KUKA KRL program: Rack_Azul_CogerST121N.src, Rack_Azul_CogerST121N.dat

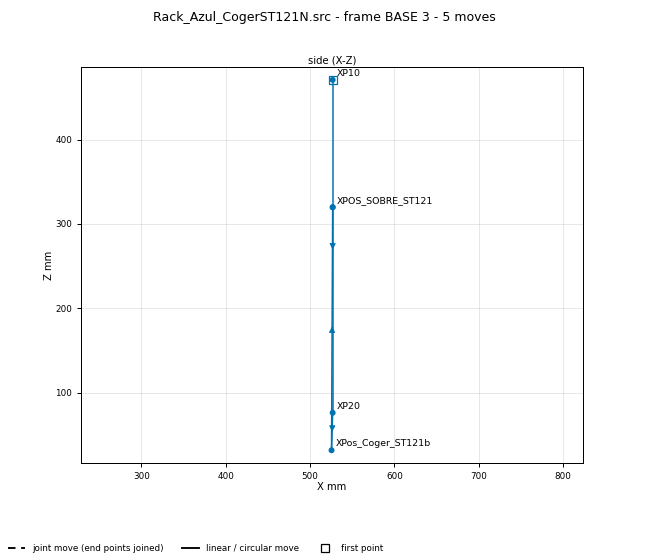
[picture p0: tool path of Rack_Azul_CogerST121N.src in frame BASE 3, 5 of 7 moves have a stored position in this frame; points joined in program order, loops and branches not executed]
--- Rack_Azul_CogerST121N.src ---
&ACCESS RVO1
&REL 24
&COMMENT COGER ST121 RACK AZUL
&PARAM EDITMASK = *
&PARAM TEMPLATE = C:\KRC\Roboter\Template\vorgabe
&PARAM DISKPATH = KRC:\R1\Program\MAFELEC
DEF Rack_Azul_CogerST121N( )
;FOLD INI;%{PE}
  ;FOLD BASISTECH INI
    GLOBAL INTERRUPT DECL 3 WHEN $STOPMESS==TRUE DO IR_STOPM ( )
    INTERRUPT ON 3
    BAS (#INITMOV,0 )
  ;ENDFOLD (BASISTECH INI)
;FOLD SPOTTECH INI
USERSPOT(#INIT)
;ENDFOLD (SPOTTECH INI)
;FOLD GRIPPERTECH INI
USER_GRP(0,DUMMY,DUMMY,GDEFAULT)
;ENDFOLD (GRIPPERTECH INI)
;FOLD USER INI
INTERRUPT DECL 26 WHEN I_121R1S102 OR I_121R1S202 DO PARO_RAPIDO ()
INTERRUPT DECL 27 WHEN I_121R1S302 OR I_121R1S402 DO PARO_RAPIDO ()

    ;Make your modifications here

  ;ENDFOLD (USER INI)
;ENDFOLD (INI)
;################################################
; PROYECTO: MAFELEC PLANTA DE BATERIAS
; ROBOT: 121_R1
; PROGRAMA: CARGA DE BATERIA EN ST121
;           POSICION DE CARGA PRODUCCION NORMAL
; CREADO POR: Alejandro Company(zaisor robotics)
; FECHA: 23-NOVIEMBRE-2022
; MODIFICADO POR:
; FECHA MODIFICACION: 13-ENERO-2023
;################################################

Empujador(1,"R",FALSE)
Empujador(2,"R",FALSE)

; FOLD ESPERA CONFIRMACION ENTRADA NORMAL
WAIT FOR NOT I_ST121_INSPECCION
; ENDFOLD

;FOLD PTP POS_ESPERA_ST121 Vel=100 % H Tool[9]:T_Gripper1_Vacio Base[0];%{PE}%R 8.3.48,%MKUKATPBASIS,%CMOVE,%VPTP,%P 1:PTP, 2:POS_ESPERA_ST121, 3:, 5:100, 7:H
$BWDSTART=FALSE
PDAT_ACT=PH
FDAT_ACT=FPOS_ESPERA_ST121
BAS(#PTP_PARAMS,100)
PTP XPOS_ESPERA_ST121
;ENDFOLD

; FOLD ESPERA CONFIRMACION ENTRADA NORMAL
WAIT FOR NOT I_ST121_INSPECCION
; ENDFOLD

; FOLD CONTROL DE MOVIMIENTOS MECANICOS EN REPOSO
;CONTROL DE AUSENCIA DE PIEZA EN GRIPPER
IF I_121R1S1000 THEN
HALT
ENDIF

;CONTROL APERTURA GRIPPER

IF (I_121R1S131B==FALSE) OR (I_121R1S132B==FALSE) OR (I_121R1S133B==FALSE) OR (I_121R1S134B==FALSE) THEN
Pines("R")
ENDIF

Empujador(1,"R",TRUE)
Empujador(2,"R",TRUE)
; ENDFOLD

;FOLD PTP P10 CONT Vel=100 % M Tool[9]:T_Gripper1_Vacio Base[3]:ST121;%{PE}%R 8.3.48,%MKUKATPBASIS,%CMOVE,%VPTP,%P 1:PTP, 2:P10, 3:C_DIS, 5:100, 7:M
$BWDSTART=FALSE
PDAT_ACT=PM
FDAT_ACT=FP10
BAS(#PTP_PARAMS,100)
PTP XP10 C_DIS
;ENDFOLD
;FOLD LIN P20 Vel=1 m/s M Tool[9]:T_Gripper1_Vacio Base[3]:ST121;%{PE}%R 8.3.48,%MKUKATPBASIS,%CMOVE,%VLIN,%P 1:LIN, 2:P20, 3:, 5:1, 7:M
$BWDSTART=FALSE
LDAT_ACT=LM
FDAT_ACT=FP20
BAS(#CP_PARAMS,1)
LIN XP20
;ENDFOLD

; FOLD ACTIVA VIGILANCIA SOBREPASO
INTERRUPT ON 26
INTERRUPT ON 27
;ENDFOLD

; POSICION DE CARGA EN ST121
;FOLD LIN Pos_Coger_ST121b Vel=0.05 m/s L Tool[9]:T_Gripper1_Vacio Base[3]:ST121;%{PE}%R 8.3.48,%MKUKATPBASIS,%CMOVE,%VLIN,%P 1:LIN, 2:Pos_Coger_ST121b, 3:, 5:0.05, 7:L
$BWDSTART=FALSE
LDAT_ACT=LL
FDAT_ACT=FPos_Coger_ST121b
BAS(#CP_PARAMS,0.05)
LIN XPos_Coger_ST121b
;ENDFOLD

; FOLD CONTROL DE PRESENCIAS PINES
Repite=0
IF (I_121R1S102==TRUE) OR (I_121R1S202==TRUE) OR (I_121R1S302==TRUE) OR (I_121R1S402==TRUE) THEN

   WHILE (I_121R1S102==TRUE) OR (I_121R1S202==TRUE) OR (I_121R1S302==TRUE) OR (I_121R1S402==TRUE)

      IF Repite>=4 THEN
         HALT
         ; SUPERADO NUMERO DE REPETICIONES
         HALT
         WAIT FOR FALSE

      ENDIF



      Repite=Repite+1
      LIN_REL{Z 1}
      WAIT SEC 0.2


   ENDWHILE
ENDIF




Repite=0
WHILE (I_121R1S101==FALSE) OR (I_121R1S201==FALSE) OR (I_121R1S301==FALSE) OR (I_121R1S401==FALSE)
IF (I_121R1S102==TRUE) OR (I_121R1S202==TRUE) OR (I_121R1S302==TRUE) OR (I_121R1S402==TRUE) THEN
HALT
HALT
HALT
ENDIF
Repite=Repite+1
LIN_REL{Z -1}
WAIT SEC 0.2

IF Repite>=5 THEN
HALT
; SUPERADO NUMERO DE REPETICIONES
HALT
ENDIF

ENDWHILE

WAIT FOR I_121R1S101 AND I_121R1S301 OR I_121R1S201 AND I_121R1S401
; ENDFOLD

Pines("A")

IF (I_SIMULACION==FALSE) THEN
WAIT FOR I_121R1S1000
ENDIF

;FIN DE TRABAJO COGER
O_JRDY_3=TRUE

; FOLD FIN VIGILANCIA SOBREPASO
INTERRUPT OFF 26
INTERRUPT OFF 27
;ENDFOLD
;FOLD TORQMON SetLimits Axis1: 50 % Axis2: 50 % Axis3: 50 % Axis4: 50 % Axis5: 50 % Axis6: 50 %;%{PE}%R 8.3.48,%MKUKATPBASIS,%CTQ_MON,%VTQ_LIMITS,%P 2:TQ_LIMITS, 4:50, 7:50, 10:50, 13:50, 16:50, 19:50
SET_TQ_VALUES (50,50,50,50,50,50)
;ENDFOLD

;FOLD LIN POS_SOBRE_ST121 Vel=0.5 m/s M Tool[11]:T_Gripper1_Carga Base[3]:ST121;%{PE}%R 8.3.48,%MKUKATPBASIS,%CMOVE,%VLIN,%P 1:LIN, 2:POS_SOBRE_ST121, 3:, 5:0.5, 7:M
$BWDSTART=FALSE
LDAT_ACT=LM
FDAT_ACT=FPOS_SOBRE_ST121
BAS(#CP_PARAMS,0.5)
LIN XPOS_SOBRE_ST121
;ENDFOLD

;FOLD TORQMON SetDefault;%{PE}%R 8.3.48,%MKUKATPBASIS,%CTQ_MON,%VTQ_DEFAULT,%P 2:TQ_DEFAULT
SET_TQ_VALUES ( )
;ENDFOLD
IF (I_SIMULACION==FALSE) THEN
WAIT FOR I_121R1S1000
ENDIF

;Revisa sensores ok antes de continuar
;FOLD WAIT FOR ( IN 253 'I_121R1_S101 PIN1 Control Pieza' );%{PE}%R 8.3.48,%MKUKATPBASIS,%CEXT_WAIT_FOR,%VEXT_WAIT_FOR,%P 2:, 4:, 5:$IN, 6:253, 7:I_121R1_S101 PIN1 Control Pieza, 9:
WAIT FOR  ( $IN[253] )
;ENDFOLD
;FOLD WAIT FOR ( NOT IN 254 'I_121R1_S102 PIN1 Sobrepaso' );%{PE}%R 8.3.48,%MKUKATPBASIS,%CEXT_WAIT_FOR,%VEXT_WAIT_FOR,%P 2:, 4:NOT, 5:$IN, 6:254, 7:I_121R1_S102 PIN1 Sobrepaso, 9:
WAIT FOR  (  NOT $IN[254] )
;ENDFOLD
;FOLD WAIT FOR ( IN 255 'I_121R1_S201 PIN2 Control Pieza' );%{PE}%R 8.3.48,%MKUKATPBASIS,%CEXT_WAIT_FOR,%VEXT_WAIT_FOR,%P 2:, 4:, 5:$IN, 6:255, 7:I_121R1_S201 PIN2 Control Pieza, 9:
WAIT FOR  ( $IN[255] )
;ENDFOLD
;FOLD WAIT FOR ( NOT IN 256 'I_121R1_S202 PIN2 Sobrepaso' );%{PE}%R 8.3.48,%MKUKATPBASIS,%CEXT_WAIT_FOR,%VEXT_WAIT_FOR,%P 2:, 4:NOT, 5:$IN, 6:256, 7:I_121R1_S202 PIN2 Sobrepaso, 9:
WAIT FOR  (  NOT $IN[256] )
;ENDFOLD
;FOLD WAIT FOR ( IN 257 'I_121R1_S301 PIN3 Control Pieza' );%{PE}%R 8.3.48,%MKUKATPBASIS,%CEXT_WAIT_FOR,%VEXT_WAIT_FOR,%P 2:, 4:, 5:$IN, 6:257, 7:I_121R1_S301 PIN3 Control Pieza, 9:
WAIT FOR  ( $IN[257] )
;ENDFOLD
;FOLD WAIT FOR ( NOT IN 258 'I_121R1_S302 PIN3 Sobrepaso' );%{PE}%R 8.3.48,%MKUKATPBASIS,%CEXT_WAIT_FOR,%VEXT_WAIT_FOR,%P 2:, 4:NOT, 5:$IN, 6:258, 7:I_121R1_S302 PIN3 Sobrepaso, 9:
WAIT FOR  (  NOT $IN[258] )
;ENDFOLD
;FOLD WAIT FOR ( IN 259 'I_121R1_S401 PIN4 Control Pieza' );%{PE}%R 8.3.48,%MKUKATPBASIS,%CEXT_WAIT_FOR,%VEXT_WAIT_FOR,%P 2:, 4:, 5:$IN, 6:259, 7:I_121R1_S401 PIN4 Control Pieza, 9:
WAIT FOR  ( $IN[259] )
;ENDFOLD
;FOLD WAIT FOR ( NOT IN 260 'I_121R1_S402 PIN4 Sobrepaso' );%{PE}%R 8.3.48,%MKUKATPBASIS,%CEXT_WAIT_FOR,%VEXT_WAIT_FOR,%P 2:, 4:NOT, 5:$IN, 6:260, 7:I_121R1_S402 PIN4 Sobrepaso, 9:
WAIT FOR  (  NOT $IN[260] )
;ENDFOLD
WAIT SEC 0.2

;FOLD PTP P30 CONT Vel=100 % L Tool[11]:T_Gripper1_Carga Base[3]:ST121;%{PE}%R 8.3.48,%MKUKATPBASIS,%CMOVE,%VPTP,%P 1:PTP, 2:P30, 3:C_DIS, 5:100, 7:L
$BWDSTART=FALSE
PDAT_ACT=PL
FDAT_ACT=FP30
BAS(#PTP_PARAMS,100)
PTP XP30 C_DIS
;ENDFOLD

;POSICION AREA 3 LIBRE
;FOLD PTP POS_AREA_3_LIBRE Vel=100 % L Tool[11]:T_Gripper1_Carga Base[0];%{PE}%R 8.3.48,%MKUKATPBASIS,%CMOVE,%VPTP,%P 1:PTP, 2:POS_AREA_3_LIBRE, 3:, 5:100, 7:L
$BWDSTART=FALSE
PDAT_ACT=PL
FDAT_ACT=FPOS_AREA_3_LIBRE
BAS(#PTP_PARAMS,100)
PTP XPOS_AREA_3_LIBRE
;ENDFOLD

;LIBERA AREA 3, TRANSPORTE BATERIAS
O_AREL_3=TRUE

WAIT FOR (I_ARDY_2) OR ($SR_RANGE_ACTIVE[16]==FALSE)
If ($SR_RANGE_ACTIVE[16]==FALSE) THEN
FromAzul2pickN()
ENDIF


END
DEF PARO_RAPIDO ()
BRAKE F
END

--- Rack_Azul_CogerST121N.dat ---
&ACCESS RVO1
&REL 24
&COMMENT COGER ST121 RACK AZUL
&PARAM EDITMASK = *
&PARAM TEMPLATE = C:\KRC\Roboter\Template\vorgabe
&PARAM DISKPATH = KRC:\R1\Program\MAFELEC
DEFDAT  Rack_Azul_CogerST121N
;FOLD EXTERNAL DECLARATIONS;%{PE}%MKUKATPBASIS,%CEXT,%VCOMMON,%P
;FOLD GRIPPERTECH EXT
EXT  H50 (INT  :IN,INT  :IN,INT  :IN,GRP_TYP  :IN )
;ENDFOLD (GRIPPERTECH EXT)
;FOLD SPOTTECH EXT
EXT  USERSPOT (S_COMMAND  :IN,SPOT_TYPE  :IN )
;ENDFOLD (SPOTTECH EXT)
;FOLD BASISTECH EXT;%{PE}%MKUKATPBASIS,%CEXT,%VEXT,%P
EXT  BAS (BAS_COMMAND  :IN,REAL  :IN )
DECL INT SUCCESS
;ENDFOLD (BASISTECH EXT)
;FOLD USER EXT;%{E}%MKUKATPUSER,%CEXT,%VEXT,%P
;Make your modifications here

;ENDFOLD (USER EXT)
;ENDFOLD (EXTERNAL DECLARATIONS)
DECL BASIS_SUGG_T LAST_BASIS={POINT1[] "Pos_Coger_ST121b        ",POINT2[] "Pos_Coger_ST121b        ",CP_PARAMS[] "L                       ",PTP_PARAMS[] "PDAT0                   ",CONT[] "                        ",CP_VEL[] "0.05                    ",PTP_VEL[] " 100                    ",SYNC_PARAMS[] "SYNCDAT                 ",SPL_NAME[] "S0                      ",A_PARAMS[] "ADAT0                   "}
DECL PDAT PH={VEL 100.000,ACC 100.000,APO_DIST 100.000,APO_MODE #CDIS,GEAR_JERK 50.0000,EXAX_IGN 0}
DECL E6POS XP10={X 526.847961,Y 673.459412,Z 470.919037,A 179.492218,B -0.271942735,C 179.783508,S 2,T 10,E1 0.0,E2 0.0,E3 0.0,E4 0.0,E5 0.0,E6 0.0}
DECL FDAT FP10={TOOL_NO 9,BASE_NO 3,IPO_FRAME #BASE,POINT2[] " ",TQ_STATE FALSE}
DECL E6POS XP20={X 526.847961,Y 674.174805,Z 76.0742,A 179.817276,B -0.271912336,C 179.783569,S 2,T 10,E1 0.0,E2 0.0,E3 0.0,E4 0.0,E5 0.0,E6 0.0}
DECL FDAT FP20={TOOL_NO 9,BASE_NO 3,IPO_FRAME #BASE,POINT2[] " ",TQ_STATE FALSE}
DECL E6POS XPOS_COGER_ST121={X 525.252,Y 674.174805,Z 32.7693672,A 179.817276,B -0.271912307,C 179.783569,S 2,T 10,E1 0.0,E2 0.0,E3 0.0,E4 0.0,E5 0.0,E6 0.0}
DECL FDAT FPos_Coger_ST121={TOOL_NO 9,BASE_NO 3,IPO_FRAME #BASE,POINT2[] " ",TQ_STATE FALSE}
DECL PDAT PM={VEL 100.000,ACC 50.0000,APO_DIST 50.0000,APO_MODE #CDIS,GEAR_JERK 50.0000,EXAX_IGN 0}
DECL E6POS XPOS_ESPERA_ST121={X 1597.05444,Y -395.116150,Z 1941.31274,A -176.307449,B 30.3077869,C -171.065643,S 2,T 10,E1 0.0,E2 0.0,E3 0.0,E4 0.0,E5 0.0,E6 0.0}
DECL FDAT FPOS_ESPERA_ST121={TOOL_NO 9,BASE_NO 0,IPO_FRAME #BASE,POINT2[] " ",TQ_STATE FALSE}
DECL LDAT LM={VEL 2.00000,ACC 25.0000,APO_DIST 100.000,APO_FAC 50.0000,AXIS_VEL 100.000,AXIS_ACC 100.000,ORI_TYP #VAR,CIRC_TYP #BASE,JERK_FAC 50.0000,GEAR_JERK 50.0000,EXAX_IGN 0}
DECL E6POS XPOS_SOBRE_ST121={X 526.847961,Y 673.459412,Z 319.874695,A 179.491791,B -0.271912426,C 179.783569,S 2,T 10,E1 0.0,E2 0.0,E3 0.0,E4 0.0,E5 0.0,E6 0.0}
DECL FDAT FPOS_SOBRE_ST121={TOOL_NO 11,BASE_NO 3,IPO_FRAME #BASE,POINT2[] " ",TQ_STATE FALSE}
DECL E6POS XPOS_SOBRE_ST122={X 1790.32410,Y 1.34322268E-13,Z 1909.62585,A -180.000,B 89.9853210,C -180.000,S 2,T 3,E1 0.0,E2 0.0,E3 0.0,E4 0.0,E5 0.0,E6 0.0}
DECL FDAT FPOS_SOBRE_ST122={TOOL_NO 9,BASE_NO 3,IPO_FRAME #BASE,POINT2[] " ",TQ_STATE FALSE}
DECL E6POS XP30={X 526.847961,Y 673.459412,Z 319.874695,A 179.491791,B -0.271912456,C 179.783569,S 2,T 10,E1 0.0,E2 0.0,E3 0.0,E4 0.0,E5 0.0,E6 0.0}
DECL FDAT FP30={TOOL_NO 11,BASE_NO 3,IPO_FRAME #BASE,POINT2[] " ",TQ_STATE FALSE}
DECL E6POS XP40={X -0.0319372341,Y -2.62910700,Z -362.053223,A -0.00123304490,B -0.0257057231,C 0.00384289422,S 2,T 10,E1 0.0,E2 0.0,E3 0.0,E4 0.0,E5 0.0,E6 0.0}
DECL FDAT FP40={TOOL_NO 11,BASE_NO 3,IPO_FRAME #BASE,POINT2[] " ",TQ_STATE FALSE}
DECL E6POS XPOS_AREA_3_LIBRE={X 1457.33850,Y 287.686401,Z 1296.45581,A 90.0126114,B -0.311890274,C -179.676559,S 2,T 43,E1 0.0,E2 0.0,E3 0.0,E4 0.0,E5 0.0,E6 0.0}
DECL FDAT FPOS_AREA_3_LIBRE={TOOL_NO 11,BASE_NO 0,IPO_FRAME #BASE,POINT2[] " ",TQ_STATE FALSE}
DECL GRP_SUGG_T LAST_GRP={NUMBER[] "1                       ",STATE[] "1                       ",PARAMS[] "GDAT0                   "}
DECL LDAT LL={VEL 2.00000,ACC 25.0000,APO_DIST 100.000,APO_FAC 50.0000,AXIS_VEL 100.000,AXIS_ACC 100.000,ORI_TYP #VAR,CIRC_TYP #BASE,JERK_FAC 50.0000,GEAR_JERK 50.0000,EXAX_IGN 0}
DECL PDAT PL={VEL 100.000,ACC 25.0000,APO_DIST 50.0000,APO_MODE #CDIS,GEAR_JERK 50.0000,EXAX_IGN 0}
DECL E6POS XPOS_COGER_ST121B={X 525.498474,Y 674.343750,Z 31.6438618,A 179.817947,B -0.451363772,C 179.783569,S 2,T 10,E1 0.0,E2 0.0,E3 0.0,E4 0.0,E5 0.0,E6 0.0}
DECL FDAT FPos_Coger_ST121b={TOOL_NO 9,BASE_NO 3,IPO_FRAME #BASE,POINT2[] " ",TQ_STATE FALSE}
ENDDAT
